FUNCTION F_StopAnalogRamping_ForRecipe
VAR
	i: UINT;
END_VAR

FOR i:= 1 TO GVL_CONSTANT.NumAnalogController DO
	GVL_IO.aController[i].input.restart := TRUE;
	GVL_IO.aController[i].input.rampTime := 1; 
	GVL_IO.aController[i].input.targetValue := LREAL_TO_REAL(GVL_IO.aController[i].rControlValue);
END_FOR

END_FUNCTION

(* stored: Version 1.1.0.1, ProductVersion 3.1.4026.12
   POU F_StopAnalogRamping_ForRecipe: Id {894f4883-78ef-41b6-90b5-91f6e5cdbce2}, SpecialFunc None *)
